// Mitsubishi GX Works2 project: 0625(연산결과뒤집기)   PLC: Q02/Q02H

PROGRAM MAIN
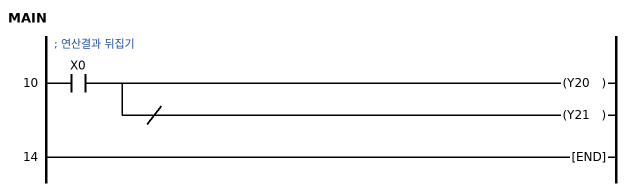
; 연산결과 뒤집기
10    LD      X0
      OUT     Y20
      INV
      OUT     Y21
14    END
END_PROGRAM
